{attribute 'qualified_only'}
VAR_GLOBAL
	stateGRAB: INT := 0;
	newStateGRAB: INT := 0;
	currentStateGRAB: INT;
	
	homingState: INT := 1;
	homingDone: BOOL := FALSE;
	
	stop: BOOL := FALSE;
END_VAR

(* stored: Version 1.1.0.1, ProductVersion 3.1.4024.6
   GVL GVL: Id {e15296e5-ac30-4ffc-ae54-f5edceddab02} *)
